FUNCTION_BLOCK ctb1
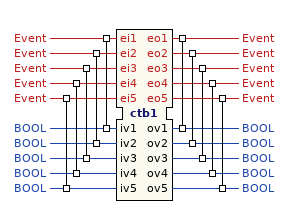
  EVENT_INPUT
    ei1 WITH iv1;
    ei2 WITH iv2;
    ei3 WITH iv3;
    ei4 WITH iv4;
    ei5 WITH iv5;
  END_EVENT
  EVENT_OUTPUT
    eo1 WITH ov1;
    eo2 WITH ov2;
    eo3 WITH ov3;
    eo4 WITH ov4;
    eo5 WITH ov5;
  END_EVENT
  VAR_INPUT
    iv1 : BOOL;
    iv2 : BOOL;
    iv3 : BOOL;
    iv4 : BOOL;
    iv5 : BOOL;
  END_VAR
  VAR_OUTPUT
    ov1 : BOOL;
    ov2 : BOOL;
    ov3 : BOOL;
    ov4 : BOOL;
    ov5 : BOOL;
  END_VAR
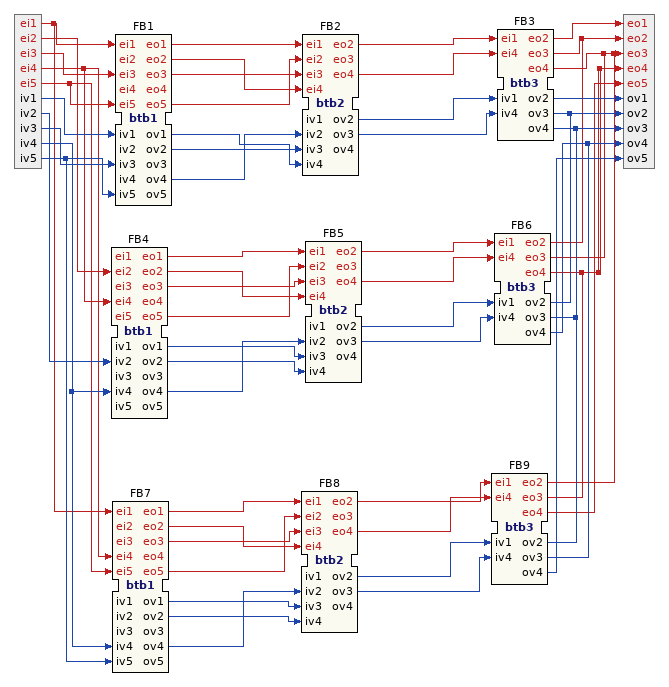
  FBS
    FB1 : btb1;
    FB2 : btb2;
    FB3 : btb3;
    FB4 : btb1;
    FB5 : btb2;
    FB6 : btb3;
    FB7 : btb1;
    FB8 : btb2;
    FB9 : btb3;
  END_FBS
  EVENT_CONNECTIONS
    ei1 TO FB1.ei1;
    ei3 TO FB1.ei3;
    ei5 TO FB1.ei5;
    ei2 TO FB4.ei2;
    ei4 TO FB4.ei4;
    ei5 TO FB7.ei5;
    ei4 TO FB7.ei4;
    ei1 TO FB7.ei1;
    FB1.eo1 TO FB2.ei1;
    FB1.eo2 TO FB2.ei4;
    FB1.eo3 TO FB2.ei3;
    FB1.eo5 TO FB2.ei2;
    FB4.eo1 TO FB5.ei1;
    FB4.eo2 TO FB5.ei4;
    FB4.eo3 TO FB5.ei3;
    FB4.eo5 TO FB5.ei2;
    FB7.eo1 TO FB8.ei1;
    FB7.eo2 TO FB8.ei4;
    FB7.eo3 TO FB8.ei3;
    FB7.eo5 TO FB8.ei2;
    FB2.eo2 TO FB3.ei1;
    FB5.eo2 TO FB6.ei1;
    FB3.eo2 TO eo1;
    FB3.eo3 TO eo2;
    FB3.eo4 TO eo3;
    FB6.eo2 TO eo2;
    FB6.eo3 TO eo3;
    FB6.eo4 TO eo4;
    FB9.eo2 TO eo3;
    FB9.eo3 TO eo4;
    FB9.eo4 TO eo5;
    FB2.eo4 TO FB3.ei4;
    FB5.eo4 TO FB6.ei4;
    FB8.eo4 TO FB9.ei4;
    FB8.eo2 TO FB9.ei1;
  END_CONNECTIONS
  DATA_CONNECTIONS
    iv1 TO FB1.iv1;
    iv3 TO FB1.iv3;
    iv5 TO FB1.iv5;
    iv2 TO FB4.iv2;
    iv4 TO FB4.iv4;
    iv5 TO FB7.iv5;
    iv4 TO FB7.iv4;
    FB1.ov4 TO FB2.iv2;
    FB1.ov2 TO FB2.iv4;
    FB1.ov1 TO FB2.iv3;
    FB4.ov4 TO FB5.iv2;
    FB4.ov2 TO FB5.iv4;
    FB4.ov1 TO FB5.iv3;
    FB7.ov4 TO FB8.iv2;
    FB7.ov2 TO FB8.iv4;
    FB7.ov1 TO FB8.iv3;
    FB2.ov2 TO FB3.iv1;
    FB5.ov2 TO FB6.iv1;
    FB8.ov2 TO FB9.iv1;
    FB3.ov2 TO ov1;
    FB3.ov3 TO ov2;
    FB3.ov4 TO ov3;
    FB6.ov2 TO ov2;
    FB6.ov3 TO ov3;
    FB6.ov4 TO ov4;
    FB9.ov2 TO ov3;
    FB9.ov3 TO ov4;
    FB9.ov4 TO ov5;
    FB2.ov3 TO FB3.iv4;
    FB5.ov3 TO FB6.iv4;
    FB8.ov3 TO FB9.iv4;
  END_CONNECTIONS
END_FUNCTION_BLOCK
